(*

short summary
=============
A specialized candy. It can be consumed by any candy consumer.
It supports dynamic creation. Furthermore, it calls the method 
AbstractCandy.initializeDispatchers after FB_init.

legal notes
===========
SPDX-FileCopyrightText: © 2024 ekvip automation GmbH <info@ekvip.de>
SPDX-License-Identifier: Apache-2.0
For details check: Apache-2.0_

.. _Apache-2.0: https://www.apache.org/licenses/LICENSE-2.0

*)

{attribute 'enable_dynamic_creation'}
{attribute 'call_after_init'}
FUNCTION_BLOCK FINAL WonkaGobstopper EXTENDS AbstractCandy
VAR_INPUT
END_VAR
VAR_OUTPUT
END_VAR
VAR
END_VAR

(*

short summary
=============
it initializes the amount, the candy name and 
the binary coded candy type  

legal notes
===========
SPDX-FileCopyrightText: © 2024 ekvip automation GmbH <info@ekvip.de>
SPDX-License-Identifier: Apache-2.0
For details check: Apache-2.0_

.. _Apache-2.0: https://www.apache.org/licenses/LICENSE-2.0

*)

METHOD FB_init :BOOL
VAR_INPUT
	(* if TRUE, the retain variables are initialized (warm start / cold start) *)
	bInitRetains	:BOOL;
	(* if TRUE, the instance afterwards gets moved into the copy code (online change) *)
	bInCopyCode		:BOOL;
END_VAR
THIS^.amount := 141;
THIS^.name := 'Wonka Gobstopper';
THIS^.candyType := CandyTypes.JAWBREAKERS OR CandyTypes.SOUR_CANDY OR CandyTypes.HARD_CANDY;
END_METHOD

END_FUNCTION_BLOCK

(* stored: Version 1.1.0.1
   POU WonkaGobstopper: Id {3e43c0ac-ea85-421e-ae49-a312a0d0c89a}, SpecialFunc None
   Method FB_init: Id {434944b9-6db4-4198-9fe3-c38e6666a9a6} *)
